SUBAPPLICATION mapping_Buttons (* Subapplication Type *)
  (* Standard: 61499-2 *)
  (* Version 1.0, 2023-01-29, Franz *)
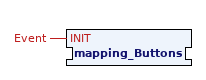
  EVENT_INPUT
    INIT;
  END_EVENT
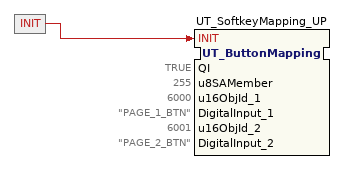
  FBS
    UT_SoftkeyMapping_UP : UT_ButtonMapping(QI := TRUE, u8SAMember := 255, u16ObjId_1 := 6000, DigitalInput_1 := "PAGE_1_BTN", u16ObjId_2 := 6001, DigitalInput_2 := "PAGE_2_BTN");
  END_FBS
  EVENT_CONNECTIONS
    INIT TO UT_SoftkeyMapping_UP.INIT;
  END_CONNECTIONS
END_SUBAPPLICATION
